// TIA Portal project "SCL_testing" (V15.1)

(* hardware
DEVICE "S71500/ET200MP station_1"  S7-1500 station
   slot 0: "Rail_0"  Rack  6ES7 590-1***0-0AA0
   slot 1: "PLC_1"  CPU 1513-1 PN  6ES7 513-1AL02-0AB0  V2.6
      slot 3: "CPU display_1"  6ES7591-1AA00-0AA0
DEVICE "HMI_1"  KTP900 Basic PN
   slot 0: "HMI_1"  KTP900 Basic PN  6AV2 123-2JB03-0AX0  15.1.0.0
   slot 1: "HMI_RT_1"  KTP900 Basic PN  6AV2 123-2JB03-0AX0  15.1.0.0
   slot 5: "HMI_1.IE_CP_1"  PROFINET Interface  15.0.1.0
      slot 1: "PROFINET Interface_1"  PROFINET Interface
         slot 1: "Port_1"  Port
*)

// ===== PLC "PLC_1"  CPU 1513-1 PN =====

VAR_GLOBAL   // PLC tag table "Default tag table"
   "Clock_Byte" AT %MB8069 : Byte;
   "Clock_10Hz" AT %M8069.0 : Bool;
   "Clock_5Hz" AT %M8069.1 : Bool;
   "Clock_2.5Hz" AT %M8069.2 : Bool;
   "Clock_2Hz" AT %M8069.3 : Bool;
   "Clock_1.25Hz" AT %M8069.4 : Bool;
   "Clock_1Hz" AT %M8069.5 : Bool;
   "Clock_0.625Hz" AT %M8069.6 : Bool;
   "Clock_0.5Hz" AT %M8069.7 : Bool;
   "System_Byte" AT %MB8080 : Byte;
   "FirstScan" AT %M8080.0 : Bool;
   "DiagStatusUpdate" AT %M8080.1 : Bool;
   "AlwaysTRUE" AT %M8080.2 : Bool;
   "AlwaysFALSE" AT %M8080.3 : Bool;
END_VAR

DATA_BLOCK "alarme"   // DB1
{ S7_Optimized_Access := 'TRUE' }
VERSION : 0.1
   VAR
      "array" : Array[0..15] of Bool;
      gather : Word;
   END_VAR
BEGIN
END_DATA_BLOCK

DATA_BLOCK "auxiliare"   // DB4
{ S7_Optimized_Access := 'TRUE' }
VERSION : 0.1
   VAR
      lim_inf : Real;
      lim_sup : Real;
   END_VAR
BEGIN
END_DATA_BLOCK

// folder: Hysteresis

DATA_BLOCK "Hysteresis_DB"   // DB2
{ S7_Optimized_Access := 'TRUE' }
VERSION : 0.1
   VAR
      temp_setpoint : Real;
      hysteresis : Real;
      temp_curenta : Real := 20.0;
      permisiune_pornire : Bool;
      arzator_pornit : Bool;
   END_VAR
BEGIN
END_DATA_BLOCK

// folder: Instante FB-uri

DATA_BLOCK "Hysteresis_DB_1"   // DB3
{ S7_Optimized_Access := 'TRUE' }
VERSION : 0.1
// stored: InstanceOfName Hysteresis
"Hysteresis"
BEGIN
END_DATA_BLOCK

// folder: (top level)

ORGANIZATION_BLOCK "Main"   // OB1, LAD, ProgramCycle
TITLE = "Main Program Sweep (Cycle)"
{ S7_Optimized_Access := 'TRUE' }
VERSION : 0.1
   VAR_INPUT
      Initial_Call : Bool;   // Initial call of this OB
      Remanence : Bool;   // =True, if remanent data are available
   END_VAR
BEGIN

REGION Network 1: gather de alarme
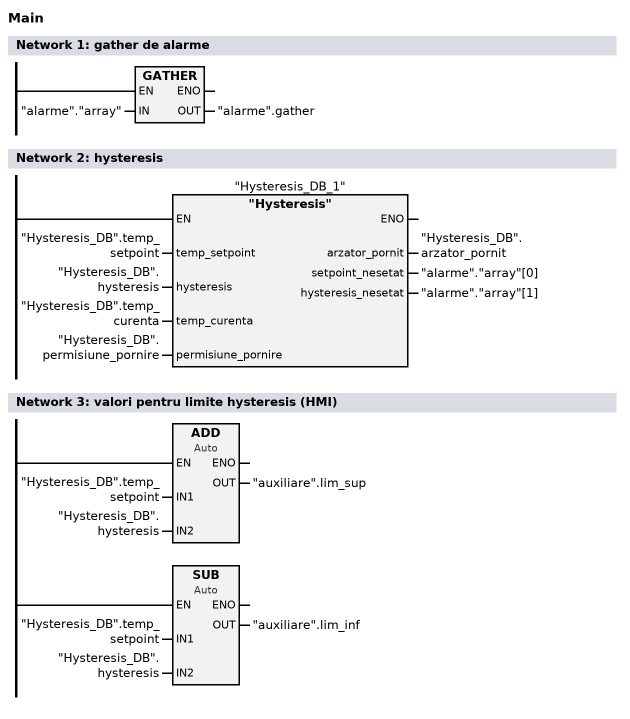
   GATHER(IN := "alarme"."array", OUT => "alarme".gather);
END_REGION

REGION Network 2: hysteresis
   RUNG wire#powerrail
      "Hysteresis_DB_1"(temp_setpoint := "Hysteresis_DB".temp_setpoint, hysteresis := "Hysteresis_DB".hysteresis, temp_curenta := "Hysteresis_DB".temp_curenta, permisiune_pornire := "Hysteresis_DB".permisiune_pornire, arzator_pornit => "Hysteresis_DB".arzator_pornit, setpoint_nesetat => "alarme"."array"[0], hysteresis_nesetat => "alarme"."array"[1])
   END_RUNG
   // the same network as SCL:
   "Hysteresis_DB_1"(temp_setpoint := "Hysteresis_DB".temp_setpoint,   // "Hysteresis"
                     hysteresis := "Hysteresis_DB".hysteresis,
                     temp_curenta := "Hysteresis_DB".temp_curenta,
                     permisiune_pornire := "Hysteresis_DB".permisiune_pornire,
                     arzator_pornit => "Hysteresis_DB".arzator_pornit,
                     setpoint_nesetat => "alarme"."array"[0],
                     hysteresis_nesetat => "alarme"."array"[1]);
END_REGION

REGION Network 3: valori pentru limite hysteresis (HMI)
   RUNG wire#powerrail
      Add(in1 := "Hysteresis_DB".temp_setpoint, in2 := "Hysteresis_DB".hysteresis, out => "auxiliare".lim_sup)
   END_RUNG
   RUNG wire#powerrail
      Sub(in1 := "Hysteresis_DB".temp_setpoint, in2 := "Hysteresis_DB".hysteresis, out => "auxiliare".lim_inf)
   END_RUNG
   // the same network as SCL:
   "auxiliare".lim_sup := "Hysteresis_DB".temp_setpoint + "Hysteresis_DB".hysteresis;
   "auxiliare".lim_inf := "Hysteresis_DB".temp_setpoint - "Hysteresis_DB".hysteresis;
END_REGION
END_ORGANIZATION_BLOCK

// folder: Hysteresis

FUNCTION_BLOCK "Hysteresis"   // FB2, LAD
{ S7_Optimized_Access := 'TRUE' }
VERSION : 0.1
   VAR_INPUT
      temp_setpoint : Real;
      hysteresis : Real;   // limitele de diferenta intre setpoint si temperatura curenta
   END_VAR
   VAR_OUTPUT
      arzator_pornit : Bool;
      setpoint_nesetat : Bool;
      hysteresis_nesetat : Bool;
   END_VAR
   VAR_IN_OUT
      temp_curenta : Real;
      permisiune_pornire : Bool;
   END_VAR
   VAR
      re1 : Bool;
      re2 : Bool;
   END_VAR
   VAR_TEMP   // added for the SCL form of the ladder/FBD networks
      _w1 : Bool;
      _w2 : Bool;
   END_VAR
BEGIN

REGION Network 1 (SCL): logica de limite pentru hysteresis
   //daca nu are permisiune de pornire de la controller, automat sa nu porneasca arzatorul

   IF #permisiune_pornire = FALSE THEN
       #arzator_pornit := FALSE;
   END_IF;

   //calculul de limite pe baza la setpoint is hysteresis
   IF #temp_curenta < #temp_setpoint - #hysteresis AND #permisiune_pornire THEN
       #arzator_pornit := TRUE;
   ELSIF #temp_curenta > #temp_setpoint + #hysteresis THEN
       #arzator_pornit := FALSE;
   END_IF;
END_REGION

REGION Network 2: simularea de temperatura
   // este putin mai simplu in ladder, folosind un positive edge trigger cu un clock de 1Hz
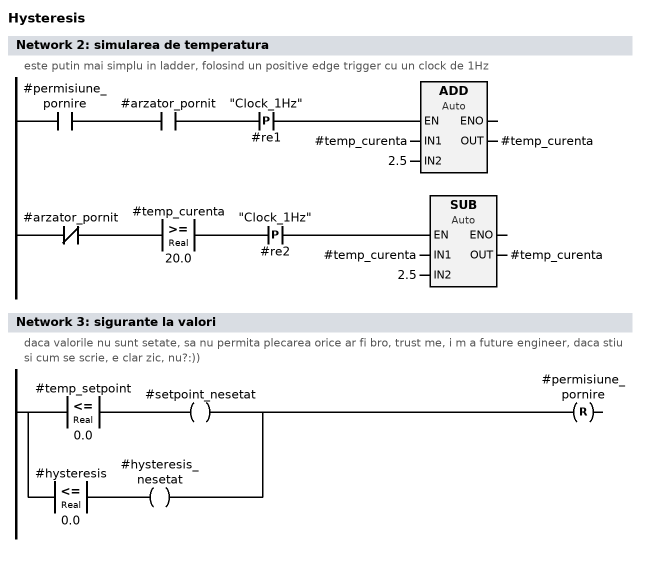
   RUNG wire#powerrail
      Contact( #permisiune_pornire )
      Contact( #arzator_pornit )
      P_Contact(operand := "Clock_1Hz", bit := #re1)
      Add(in1 := #temp_curenta, in2 := 2.5, out => #temp_curenta)
   END_RUNG
   RUNG wire#powerrail
      I_Contact( #arzator_pornit )
      { S7_Templates := "SrcType := Real" } GE_Contact(in1 := #temp_curenta, in2 := 20.0)
      P_Contact(operand := "Clock_1Hz", bit := #re2)
      Sub(in1 := #temp_curenta, in2 := 2.5, out => #temp_curenta)
   END_RUNG
   // the same network as SCL:
   #_w1 := #permisiune_pornire AND #arzator_pornit AND "Clock_1Hz" AND NOT #re1;   // rising edge of "Clock_1Hz"
   #re1 := "Clock_1Hz";
   IF #_w1 THEN #temp_curenta := #temp_curenta + 2.5; END_IF;
   #_w2 := NOT #arzator_pornit AND (#temp_curenta >= 20.0) AND "Clock_1Hz" AND NOT #re2;   // rising edge of "Clock_1Hz"
   #re2 := "Clock_1Hz";
   IF #_w2 THEN #temp_curenta := #temp_curenta - 2.5; END_IF;
END_REGION

REGION Network 3: sigurante la valori
   // daca valorile nu sunt setate, sa nu permita plecarea orice ar fi bro, trust me, i m a future engineer, daca stiu si cum se scrie, e clar zic, nu?:))
   RUNG wire#powerrail
      { S7_Templates := "SrcType := Real" } LE_Contact(in1 := #temp_setpoint, in2 := 0.0)
      Coil( #setpoint_nesetat )
      wire#w1
      R_Coil( #permisiune_pornire )
   END_RUNG
   RUNG wire#powerrail
      { S7_Templates := "SrcType := Real" } LE_Contact(in1 := #hysteresis, in2 := 0.0)
      Coil( #hysteresis_nesetat )
   END_RUNG wire#w1
   // the same network as SCL:
   #setpoint_nesetat := #temp_setpoint <= 0.0;
   #hysteresis_nesetat := #hysteresis <= 0.0;
   IF #setpoint_nesetat OR #hysteresis_nesetat THEN #permisiune_pornire := FALSE; END_IF;
END_REGION
END_FUNCTION_BLOCK

(* ===== HMI "HMI_RT_1" =====
system functions are stored by id; their names below are inferred from use
connection "HMI_Connection_1": ETHERNET, SMART_S7_1500_OMS

HMI tags "Default tag table"
   "alarme_gather" : Word = PLC alarme.gather, 1 s
   "Hysteresis_DB_temp_setpoint" : Real = PLC Hysteresis_DB.temp_setpoint, 1 s
   "Hysteresis_DB_hysteresis" : Real = PLC Hysteresis_DB.hysteresis, 1 s
   "Hysteresis_DB_temp_curenta" : Real = PLC Hysteresis_DB.temp_curenta, 1 s
   "Hysteresis_DB_permisiune_pornire" : Bool = PLC Hysteresis_DB.permisiune_pornire, 1 s
   "Hysteresis_DB_arzator_pornit" : Bool = PLC Hysteresis_DB.arzator_pornit, 1 s
   "auxiliare_lim_inf" : Real = PLC auxiliare.lim_inf, 1 s
   "auxiliare_lim_sup" : Real = PLC auxiliare.lim_sup, 1 s

discrete alarms
   1: 'Setpointul nu este setat', class Errors, trigger "alarme_gather" bit 0
   2: 'Hyteresis nu este setat', class Errors, trigger "alarme_gather" bit 1

screen "Main" 800x480
   IOField "I/O field_1" at 96,31 size 74x27; FormatPattern 999.99; Unit °C
      ProcessValue <- "Hysteresis_DB_temp_setpoint"
   TrendView "Trend view_1" at 218,191 size 582x288
   TextField "Text field_1" at 26,33 size 65x20; Text 'Setpoint:'
   IOField "I/O field_2" at 109,73 size 74x27; FormatPattern 999.99; Unit °C
      ProcessValue <- "Hysteresis_DB_hysteresis"
   TextField "Text field_2" at 26,75 size 79x20; Text 'Hysteresis:'
   IOField "I/O field_3" at 135,115 size 74x27; FormatPattern 999.99; Unit °C
      ProcessValue <- "Hysteresis_DB_temp_curenta"
   TextField "Text field_3" at 26,117 size 103x20; Text 'Temp. curenta:'
   Button "Button_1" at 28,162 size 69x32; TextOff 'Pornire'
      Appearance <- "Hysteresis_DB_permisiune_pornire"
      on Press: SetBit("Hysteresis_DB_permisiune_pornire")
   Circle "Circle_1" at 107,211 size 40x40
      Appearance <- "Hysteresis_DB_arzator_pornit"
   TextField "Text field_4" at 32,220 size 61x20; Text 'Arzator:'
   Button "Button_2" at 105,162 size 69x32; TextOff 'Oprire'
      on Press: ResetBit("Hysteresis_DB_permisiune_pornire")
      Appearance <- "Hysteresis_DB_permisiune_pornire"
   Button "Button_3" at 659,20 size 56x32; TextOff 'Login'
      on Press: function_a2a04561()
   Button "Button_4" at 723,20 size 56x32; TextOff 'Log off'
      on Press: function_f23ef4c9()
*)